INTERFACE I_Event EXTENDS I_Object

METHOD PUBLIC M_Debug : BOOL
VAR_INPUT
	Message:				STRING(255);
END_VAR
END_METHOD

METHOD PUBLIC M_Error : BOOL
VAR_INPUT
	Message:				STRING(255);
	ID:						UDINT;
	Severity:				E_Severity;
END_VAR
END_METHOD

METHOD PUBLIC M_Information : BOOL
VAR_INPUT
	Message:				STRING(255);
	ID:						UDINT;
END_VAR
END_METHOD

METHOD PUBLIC M_Warning : BOOL
VAR_INPUT
	Message:				STRING(255);
	ID:						UDINT;
END_VAR
END_METHOD

PROPERTY PUBLIC P_Logger : I_Logger
GET
END_GET
SET
END_SET
END_PROPERTY

END_INTERFACE

(* stored: Version 1.1.0.1
   Itf I_Event: Id {86200139-fcb7-4d9e-9f1b-6b3e88f31cc6}
   Method M_Debug: Id {de8efd53-16f5-0334-02e3-fdd0e4bf084c}
   Method M_Error: Id {7ce1cd66-528d-482d-8b65-9ae3dbff679e}
   Method M_Information: Id {a0df6aac-21ac-0b65-3426-2421a14ee702}
   Method M_Warning: Id {ae861465-4d88-0ffb-03b6-6d69b34da892}
   Property P_Logger: Id {79c5886e-8d4f-463a-a8f3-e7a7286bafb7}
   Get Get: Id {d72a2fbe-a299-4aee-94b4-9d545177e15c}
   Set Set: Id {769c2202-eaa4-4a8d-ad42-86a0c8601e68} *)
